FUNCTION_BLOCK FB_WS_Input
VAR_INPUT
	KL_Wetterstation_group_0_0_1	: EIB_GROUP_ADDR;
END_VAR
VAR_OUTPUT
	Windgeschwindigkeit			: REAL;
	Aussentemperatur			: REAL;
	Aussentemperatur_gemittelt	: REAL;
	Daemmerung					: REAL;
	Regensensor					: BOOL;
END_VAR
VAR
	Konvertierung 			: FB_WS_Konvertierung;
	Initialisierung			: FB_WS_Init;
	Mittelung 				: FB_WS_Mittelung;
	Impuls					: TP;
	Flanken: BOOL:=FALSE;
END_VAR

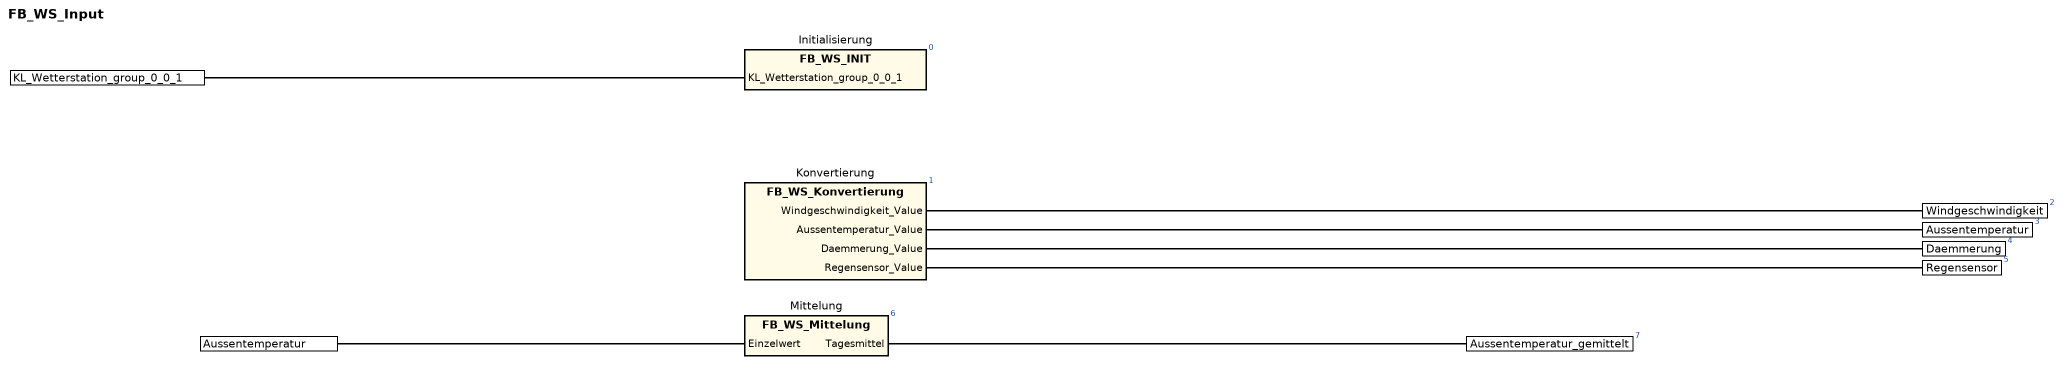
Initialisierung(KL_Wetterstation_group_0_0_1 := KL_Wetterstation_group_0_0_1); // FB_WS_INIT
Konvertierung(); // FB_WS_Konvertierung
Windgeschwindigkeit := Konvertierung.Windgeschwindigkeit_Value;
Aussentemperatur := Konvertierung.Aussentemperatur_Value;
Daemmerung := Konvertierung.Daemmerung_Value;
Regensensor := Konvertierung.Regensensor_Value;
Mittelung(Einzelwert := Aussentemperatur); // FB_WS_Mittelung
Aussentemperatur_gemittelt := Mittelung.Tagesmittel;

END_FUNCTION_BLOCK

(* stored: Version 1.1.0.1, ProductVersion 3.1.4024.9
   POU FB_WS_Input: Id {672ecb7f-9e62-4558-a118-772ead6f00bb}, SpecialFunc None *)
